Universal Robots PolyScope program: program3.urp

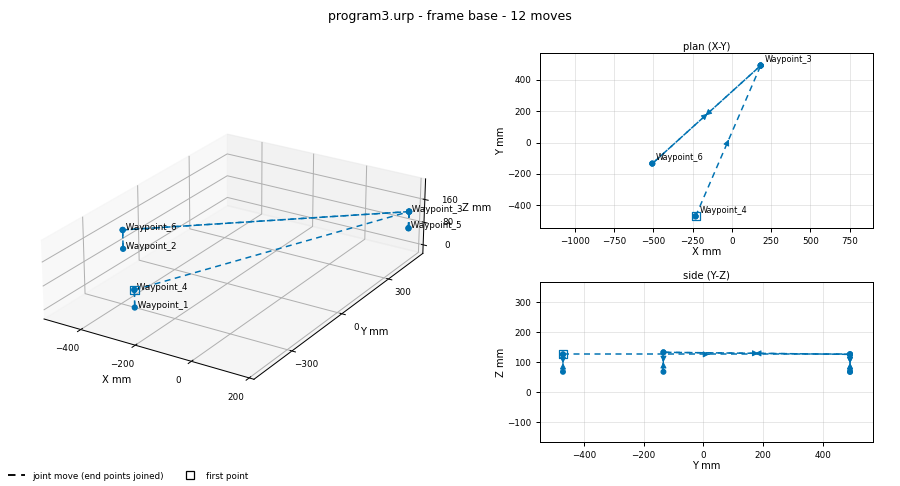
[picture p0: tool path of program3.urp in frame base, 12 of 12 moves have a stored position in this frame; points joined in program order, loops and branches not executed]
Program program3 (installation=default directory=/ursim/programs createdIn=3.15.8.106339 lastSavedIn=3.15.8.106339 robotSerialNumber=2018359999)
Calibrated DH parameters: a=[0, -0.425, -0.39225, 0, 0, 0]; d=[0.089159, 0, 0, 0.10915, 0.09465, 0.0823]; alpha=[1.570796, 0, 0, 1.570796, -1.570796, 0]; deltaTheta=[0, 0, 0, 0, 0, 0]
Robot Program (runOnlyOnce=false)
  MoveJ speed 60 deg/s, acceleration 80 deg/s^2 (useActiveTCP=true)
    Waypoint Waypoint_4: TCP in base x=-230.376 y=-469.771 z=126.472 mm, rx=-0.1122 ry=-1.5924 rz=-0.1385 rad; joints [-94.692, -113.756, -107.615, -121.526, 4.642, -288.118] deg
    Waypoint Waypoint_1: TCP in base x=-230.376 y=-469.771 z=68.074 mm, rx=-0.1122 ry=-1.5924 rz=-0.1385 rad; joints [-94.692, -119.676, -109.745, -113.476, 4.642, -288.118] deg
    Set DigitalOutput pin=digital_out[0]; digitalValue=1
    Wait Sleep waitTime=2
    Waypoint Waypoint_4: TCP in base x=-230.376 y=-469.771 z=126.472 mm, rx=-0.1122 ry=-1.5924 rz=-0.1385 rad; joints [-94.692, -113.756, -107.615, -121.526, 4.642, -288.118] deg
    Waypoint Waypoint_3: TCP in base x=183.886 y=489.84 z=126.472 mm, rx=2.2075 ry=-0.0484 rz=2.1543 rad; joints [90.856, -113.756, -107.615, -121.526, 4.642, -288.118] deg
    Waypoint Waypoint_5: TCP in base x=183.848 y=489.855 z=68.074 mm, rx=2.2076 ry=-0.0483 rz=2.1544 rad; joints [90.86, -119.676, -109.745, -113.476, 4.642, -288.118] deg
    Wait Sleep waitTime=2
  Set DigitalOutput pin=digital_out[0]; digitalValue=0
  MoveJ speed 60 deg/s, acceleration 80 deg/s^2 (useActiveTCP=true)
    Waypoint Waypoint_3: TCP in base x=183.886 y=489.84 z=126.472 mm, rx=2.2075 ry=-0.0484 rz=2.1543 rad; joints [90.856, -113.756, -107.615, -121.526, 4.642, -288.118] deg
    Waypoint Waypoint_6: TCP in base x=-505.788 y=-133.926 z=133.273 mm, rx=-0.7904 ry=-1.4525 rz=-0.7981 rad; joints [-143.737, -113.127, -107.289, -122.482, 4.642, -288.118] deg
    Waypoint Waypoint_2: TCP in base x=-505.788 y=-133.926 z=68.074 mm, rx=-0.7904 ry=-1.4525 rz=-0.7981 rad; joints [-143.737, -119.676, -109.745, -113.476, 4.642, -288.118] deg
    Wait Sleep waitTime=2
    Set DigitalOutput pin=digital_out[0]; digitalValue=1
    Waypoint Waypoint_6: TCP in base x=-505.788 y=-133.926 z=133.273 mm, rx=-0.7904 ry=-1.4525 rz=-0.7981 rad; joints [-143.737, -113.127, -107.289, -122.482, 4.642, -288.118] deg
    Waypoint Waypoint_3: TCP in base x=183.886 y=489.84 z=126.472 mm, rx=2.2075 ry=-0.0484 rz=2.1543 rad; joints [90.856, -113.756, -107.615, -121.526, 4.642, -288.118] deg
    Waypoint Waypoint_5: TCP in base x=183.848 y=489.855 z=68.074 mm, rx=2.2076 ry=-0.0483 rz=2.1544 rad; joints [90.86, -119.676, -109.745, -113.476, 4.642, -288.118] deg
    Wait Sleep waitTime=2
    Set DigitalOutput pin=digital_out[0]; digitalValue=0
    Waypoint Waypoint_3: TCP in base x=183.886 y=489.84 z=126.472 mm, rx=2.2075 ry=-0.0484 rz=2.1543 rad; joints [90.856, -113.756, -107.615, -121.526, 4.642, -288.118] deg
    Wait DigitalInput pin=digital_in[0]; digitalValue=1
